// TIA Portal V19 export
FUNCTION "SIGNAL FROM UHT" : Void   // FC25, STL
TITLE = TEST START / STOP FILLING
{ S7_Optimized_Access := 'TRUE' }
NAME : CFILLING
VERSION : 0.0
// Comment
// stored: AutoNumber false
BEGIN

NETWORK
TITLE = TEST START / STOP FILLING
// Comment
      AN    "S0 PRODUCTION TANK";
      R     "DUMMY PRODUCT AT TANK";
      BEC;
      A     "DUMMY PRODUCT AT TANK";
      JC    M001;
      AN    "OPEN_TANK";  //SIGNAL "PRODUCT AT TANK", MPI FROM UHT OR INPUT
      AN    "R.PROD  AT TANK";
      BEC;
      S     "DUMMY PRODUCT AT TANK";
      S     "START FILLING TANK";
      BEU;
M001: A     "OPEN_TANK";  //SIGNAL "PRODUCT AT TANK", MPI FROM UHT OR INPUT
      O     "R.PROD  AT TANK";
      BEC;
      R     "DUMMY PRODUCT AT TANK";
      S     "STOP FILLING TANK";
      BEU;
END_FUNCTION
